INTERFACE IPiperModule EXTENDS IPlugin
// Copyright (c) 2024 Loupe (https://loupe.team), provided under the MIT License.

METHOD Aborting : MACHINE_STATE
END_METHOD

METHOD AbortingAsync : MACHINE_STATE
END_METHOD

METHOD Booting : MACHINE_STATE
END_METHOD

METHOD BootingAsync : MACHINE_STATE
END_METHOD

METHOD CallState : BOOL
VAR_INPUT

END_VAR
END_METHOD

METHOD CallStateAsync : BOOL
VAR_INPUT
END_VAR
END_METHOD

METHOD Clearing : MACHINE_STATE
END_METHOD

METHOD ClearingAsync : MACHINE_STATE
END_METHOD

METHOD Completing : MACHINE_STATE
END_METHOD

METHOD CompletingAsync : MACHINE_STATE
END_METHOD

PROPERTY currentState : MACHINE_STATE
GET
END_GET
END_PROPERTY

METHOD didCall : BOOL
VAR_INPUT
END_VAR
END_METHOD

METHOD didCallAsync : BOOL
VAR_INPUT
END_VAR
END_METHOD

METHOD Executing : MACHINE_STATE
END_METHOD

METHOD ExecutingAsync : MACHINE_STATE
END_METHOD

METHOD Holding : MACHINE_STATE
END_METHOD

METHOD HoldingAsync : MACHINE_STATE
END_METHOD

METHOD RegisterToMachine : DINT
VAR_INPUT
    machineIn : REFERENCE TO Piper;
END_VAR
END_METHOD

{warning 'add property implementation'}
PROPERTY requestedSubstate : ULINT
GET
END_GET
END_PROPERTY

METHOD Resetting : BOOL
END_METHOD

METHOD ResettingAsync : BOOL
END_METHOD

PROPERTY response : RESPONSE_STATE
GET
END_GET
END_PROPERTY

METHOD Run : BOOL
END_METHOD

METHOD setContext : BOOL
VAR_INPUT
    context : IPluginRunner;
END_VAR
END_METHOD

METHOD setState : BOOL
VAR_INPUT
END_VAR
END_METHOD

METHOD Starting : MACHINE_STATE
END_METHOD

METHOD StartingAsync : MACHINE_STATE
END_METHOD

METHOD Stopping : MACHINE_STATE
END_METHOD

METHOD StoppingAsync : MACHINE_STATE
END_METHOD

METHOD Suspending : MACHINE_STATE
END_METHOD

METHOD SuspendingAsync : MACHINE_STATE
END_METHOD

METHOD Undefined : MACHINE_STATE
END_METHOD

METHOD UndefinedAsync : MACHINE_STATE
END_METHOD

METHOD Unholding : MACHINE_STATE
END_METHOD

METHOD UnholdingAsync : MACHINE_STATE
END_METHOD

METHOD Unsuspending : MACHINE_STATE
END_METHOD

METHOD UnsuspendingAsync : MACHINE_STATE
END_METHOD

METHOD willCall : BOOL
VAR_INPUT
END_VAR
END_METHOD

METHOD willCallAsync : BOOL
VAR_INPUT
END_VAR
END_METHOD

END_INTERFACE

(* stored: Version 1.1.0.1
   Itf IPiperModule: Id {89fd7065-3943-4b1c-ad3e-14ab7dd60316}
   Folder Handshake: Id {bfeb6266-89a6-4954-9a8c-11f58790206b}
   Folder PackML: Id {1c1d730d-e92c-4434-bb9f-84b4c155a076}
   Folder PackMLAsync: Id {ec4ba5bf-12eb-47b8-8044-3c4f8b199ed3}
   Folder setup: Id {c2d41e69-f75d-4e21-b18b-c749de73c614}
   Method Aborting: Id {31bef660-7729-4f0b-ac59-99d5c11ccaec}
   Method AbortingAsync: Id {792c629d-6eb9-4ab8-aee4-debd4d726b86}
   Method Booting: Id {5c590115-8821-4087-9459-bebd4857736c}
   Method BootingAsync: Id {5120c67c-31df-4ee9-b971-f4a960883a43}
   Method CallState: Id {547db319-98cd-43be-bfbc-09df5283103d}
   Method CallStateAsync: Id {4b455c8b-4697-405e-864a-681481284628}
   Method Clearing: Id {3d85cf08-da19-4f17-a03d-5b6ca6353df3}
   Method ClearingAsync: Id {53cb887a-8205-4038-b50a-d8035f116945}
   Method Completing: Id {5d63d193-371d-4cce-80ad-66b121f5e813}
   Method CompletingAsync: Id {102f0603-dd1d-43d8-9886-3e79acfb035d}
   Property currentState: Id {ab1ec822-8393-4376-afb7-1a080b29213a}
   Get Get: Id {0ead9c91-a998-4249-a9e9-14d3affaefd4}
   Method didCall: Id {0a5ed2d3-ceec-4a1f-a4b3-cf86c78200f7}
   Method didCallAsync: Id {4e8a607c-e9e9-49a8-b79b-39c3eddd23ea}
   Method Executing: Id {5904b031-ee1c-4c03-afef-7802b2ddbbc3}
   Method ExecutingAsync: Id {f57a4d8c-15d8-44a9-b9ef-feae480c11f5}
   Method Holding: Id {09427e55-2fcc-44f0-9fbe-8273e4905b47}
   Method HoldingAsync: Id {c5281f45-f5db-43d7-a98b-202f08f83a60}
   Method RegisterToMachine: Id {22393572-a1b0-41ae-8f7d-0c9e9c9d1a74}
   Property requestedSubstate: Id {e2364936-16e8-4c1a-b284-038a93d87878}
   Get Get: Id {ec101671-53eb-4978-b1ae-a023af1dd40c}
   Method Resetting: Id {e9dc57fb-9add-4507-941d-9416a76a3b34}
   Method ResettingAsync: Id {70243386-61db-41a6-a658-e57a3e14904f}
   Property response: Id {5aee3df5-854d-4946-a55e-2d702773392a}
   Get Get: Id {17a9ae0e-bc4f-4aa6-9d7a-68951e95c80f}
   Method Run: Id {363dda8d-c7e0-4fdc-a632-d3670d4cae33}
   Method setContext: Id {41d302b7-09fc-495b-b347-af87fcdc1c1a}
   Method setState: Id {bb8b2352-cd8c-4e74-af69-ee7d09ca216b}
   Method Starting: Id {5a22a6a4-4a12-4d54-94bf-32a7fe719ebb}
   Method StartingAsync: Id {ecc677b1-de59-417d-9106-54d979b52a4f}
   Method Stopping: Id {65bd1fc8-cdd8-4da5-b2a2-e12daa25607d}
   Method StoppingAsync: Id {a8cd60f9-a464-40bd-8146-d878194ba8d4}
   Method Suspending: Id {228751f1-bef7-4f6f-b15b-25c639455aa6}
   Method SuspendingAsync: Id {ebc3e7b0-0b95-424a-b76e-760248d5a9ce}
   Method Undefined: Id {cb777a00-4074-479f-808b-dc80a6d500a8}
   Method UndefinedAsync: Id {d4d0f36c-b93f-4f2c-bc0d-292489dcda25}
   Method Unholding: Id {c2721932-b092-4e90-881f-95da5a1389c0}
   Method UnholdingAsync: Id {2f5d526d-825d-4742-88cd-11d652b43e0d}
   Method Unsuspending: Id {89bb72a2-01ef-4f94-bb39-b3030006b691}
   Method UnsuspendingAsync: Id {ac9381ab-eb6c-4fda-8d70-0715464659c2}
   Method willCall: Id {e0e884c0-97fa-4141-a8b6-fcf6a274136a}
   Method willCallAsync: Id {44fa5592-9dbd-464e-bbb5-38e9bc21a877} *)
